// TIA Portal V20 export
TYPE "MABS_Parameters"
// stored: Namespace LineD1
   STRUCT
      StartUpTime : Time := T#5S;
      CrossSensorFilterTime : Array[1..2] of Time;
      SensorBlockageTime : Time := T#5S;
      EnergySaveTime : Time := T#4s;
   END_STRUCT;
END_TYPE
